(****************************************************************
NAME:			FB_SetPhaseLowerAxisPosition
DATA:			2022.10.18
VERSION:		1.0.0
DESCRIPTION:	FB_SetPhaseLowerAxisPosition
HISTORY:
				2022.10.18		NEW

***************************************************************)
FUNCTION_BLOCK FB_SetPhaseLowerAxisPosition
VAR_INPUT
	ValueSet:LREAL:=0;
	Execute:BOOL;
END_VAR
VAR_OUTPUT
	FbID:DINT:=1001;
	State:DINT;
	Busy:BOOL;
	Done:BOOL;
	Error:BOOL;
	ErrorID:DINT;
END_VAR
VAR
	PhaseLowerLin_MC_SetPosition: MC_SetPosition;
	fb_ton: TON;
	FB_PlcEmergencyStop: FB_PlcEmergencyStop;
END_VAR

IF Execute THEN
Busy:=TRUE;
Done:=FALSE;
fb_ton(PT:=t#0.1s);
CASE State OF
	0:
		IF PhaseLowerLin_MC_SetPosition.Error THEN		(*FB Error*)
			ErrorID:=1;
			State:=99;
		ELSE
			State:=1;
		END_IF
	1:	(*Execute*)
		PhaseLowerLin_MC_SetPosition.Position:=ValueSet;
		PhaseLowerLin_MC_SetPosition.Execute:=TRUE;
		A_SetPhaseLowerPositionMC();
		fb_ton.IN:=TRUE;
		State:=2;
	2:	(*Wait*)
		A_SetPhaseLowerPositionMC();
		IF NOT PhaseLowerLin_MC_SetPosition.Done THEN		
			IF NOT fb_ton.Q THEN
				State:=2;
			ELSE
				ErrorID:=4;
				State:=99;
			END_IF
		ELSIF  PhaseLowerLin_MC_SetPosition.Done THEN	
			State:=88;
		ELSE
			ErrorID:=5;
			State:=99;
		END_IF
	88:
		Execute:=FALSE;
		State:=0;
		Busy:=FALSE;
		Done:=TRUE;
		Error:=FALSE;
		ErrorID:=0;
		PhaseLowerLin_MC_SetPosition.Execute:=FALSE;
		fb_ton.IN:=FALSE;
	99:
		Execute:=FALSE;
		State:=99;
		Busy:=FALSE;
		Done:=FALSE;
		Error:=TRUE;
		PhaseLowerLin_MC_SetPosition.Execute:=FALSE;
		fb_ton.IN:=FALSE;
	-100:
		FB_PlcEmergencyStop();
		Execute:=FALSE;
		State:=-100;
		Busy:=FALSE;
		Done:=FALSE;
		Error:=TRUE;
		PhaseLowerLin_MC_SetPosition.Execute:=FALSE;
		fb_ton.IN:=FALSE;
END_CASE
END_IF

ACTION A_SetPhaseLowerPositionMC:
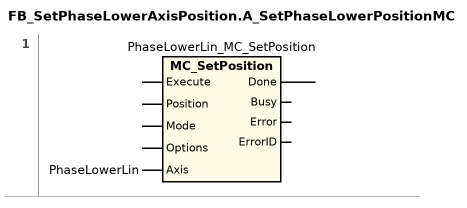
// NETWORK 1
PhaseLowerLin_MC_SetPosition(Axis := PhaseLowerLin); // MC_SetPosition
END_ACTION

END_FUNCTION_BLOCK

(* stored: Version 1.1.0.1, ProductVersion 3.1.4024.6
   POU FB_SetPhaseLowerAxisPosition: Id {5017d07c-f8cc-4ab0-bce2-987568036420}, SpecialFunc None
   Action A_SetPhaseLowerPositionMC: Id {8c120a3c-dfea-40e4-9675-3ae43a82db84} *)
